(* IEC 61131-3 sources: mastertool-rankine-bridge/tests/fixtures/sample_pous, 1 file *)

(* ---- FB_Valvula.declaration.st ---- *)
FUNCTION_BLOCK FB_Valvula EXTENDS FB_EquipamentoBase
VAR_INPUT
    xAbrir      : BOOL;
    tTimeout    : TIME := T#5S;
END_VAR
VAR_OUTPUT
    xAberta     : BOOL;
    xErro       : BOOL;
END_VAR
VAR_IN_OUT
    stComando   : ST_ComandoValvula;
END_VAR
VAR PERSISTENT
    iAcionamentos : UDINT;
END_VAR
